// TIA Portal V17 export
// export: Created 2024-01-30T08:49:17.3849629Z, ExportSetting WithDefaults, DisplayName Totally Integrated Automation Portal, DisplayVersion V17 Update 6, DisplayName TIA Portal Openness, DisplayVersion V17 Update 6, DisplayName TIA Portal Version Control Interface, DisplayVersion V17, DisplayName STEP 7 Professional, DisplayVersion V17 Update 6, DisplayName STEP 7 Safety, DisplayVersion V17 Update 6, DisplayName WinCC Advanced, DisplayVersion V17 Update 6
TYPE "UDT_LKG5000_RS232_RCV"
// stored: IsFailsafeCompliant false
   STRUCT
      Sender_ready : Bool;
      Recv_confirm : Bool;
      Frame_Error : Bool;
      ParityorSize_Error : Bool;
      Save_Overload : Bool;
      Timeout : Bool;
      Invalid_sendSize : Bool;
      Invalid_recvSize : Bool;
      Reserve : Byte;
      Recv_FrameSize : USInt;
   END_STRUCT;
END_TYPE
